PROGRAM P_Trappe_T1
VAR
	bDigitalPir				AT%I*	: BOOL;
	bTrappelysNC		AT%Q*	: BOOL;
	
	fbTon_Off				: TON;
	tPirTidOff				: TIME;
	tPirTidOff_PLC	: TIME := T#1M;
	bIngenAktivitet		: BOOL;
	bTrappeLys			: BOOL;
	
	//Modbus data Read
	bTrappeAktivitet		: BOOL;
	//Modbus data Read/Wrtite
	bPirTidOff_MB			: TIME;
	
END_VAR


bIngenAktivitet	:= NOT bDigitalPir;
tPirTidOff		:= tPirTidOff_PLC;

fbTon_Off(IN:= bIngenAktivitet, PT:= tPirTidOff);

IF bDigitalPir  THEN
	bTrappeLys := TRUE;
END_IF
IF fbTon_Off.Q THEN
	bTrappeLys := FALSE;
END_IF

bTrappelysNC 	:= NOT bTrappeLys;

END_PROGRAM

(* stored: Version 1.1.0.1
   POU P_Trappe_T1: Id {ca40d73b-b82e-4d71-9495-9c416cd53bfa}, SpecialFunc None *)
